			LogMsg := CONCAT('|CompId: ', WORD_TO_STRING(WsCfg.wCompId));
			LogMsg := CONCAT(LogMsg, '|WsNum: ');
			LogMsg := CONCAT(LogMsg, UINT_TO_STRING(WsCfg.iWsNum));
			LogMsg := CONCAT(LogMsg, '|Next State: ');
			LogMsg := CONCAT(LogMsg, UINT_TO_STRING(NextState));
			LogMsg := CONCAT(LogMsg,'|Cycle finished with Doc in Ws');
			Logging.Debug('FB_WsFsm.M_FinishCycle', LogMsg);	
		END_IF
	ELSIF NOT bProcessDocInWs THEN								//No document was processed before
		//switch to next state
			NextState := eWsStates.IDLE;
		IF GVL_Statemachine_ERROR_IDS.bLoggingOnOff THEN	
			LogMsg := CONCAT('|CompId: ', WORD_TO_STRING(WsCfg.wCompId));
			LogMsg := CONCAT(LogMsg, '|WsNum: ');
			LogMsg := CONCAT(LogMsg, UINT_TO_STRING(WsCfg.iWsNum));
			LogMsg := CONCAT(LogMsg, '|Next State: ');
			LogMsg := CONCAT(LogMsg, UINT_TO_STRING(NextState));
			LogMsg := CONCAT(LogMsg,'|Cycle finished without Doc in Ws');
			Logging.Debug('FB_WsFsm.M_FinishCycle', LogMsg);	
		END_IF
	ELSE														//wrong parameter Error	
		
		bMethodError := TRUE;
		
		//Throw Error		
			MethodErrorMsg.wErrorNo := GVL_Statemachine_ERROR_IDS.ERR_FSM_WRONG_INPUT_PARAMETER + GVL_Statemachine_ERROR_IDS.iErrorOffset;
			MethodErrorMsg.ErrorTyp	:= eErrorTypes._FATAL;
			M_ThrowError(	SrcState := CurrentState,
							ErrorMsg := MethodErrorMsg);	
		
		//Switch to Error state
			NextState := eWsStates.ERROR;				
	END_IF
ELSE		
		bMethodError:=TRUE;
		NextState := eWsStates.ERROR;
		
		MethodErrorMsg.wErrorNo := GVL_Statemachine_ERROR_IDS.ERR_FSM_WRONG_STATE_TO_FINISH_CYCLE + GVL_Statemachine_ERROR_IDS.iErrorOffset;
		MethodErrorMsg.ErrorTyp	:= eErrorTypes._FATAL;
		M_ThrowError(	SrcState := CurrentState,
						ErrorMsg := MethodErrorMsg);	
					
END_IF	
	
M_FinishCycle := bMethodError;
END_METHOD

METHOD PUBLIC M_ResetWs
VAR 
	LogMsg : STRING ;
END_VAR
(*
IF CurrentState <> eWsStates.IDLE THEN
	bisError := TRUE;
	bIsReset := TRUE;

END_IF
*)	
IF GVL_Statemachine_ERROR_IDS.bLoggingOnOff THEN	
	//Log data
		LogMsg := CONCAT('|CompId: ', WORD_TO_STRING(WsCfg.wCompId));
		LogMsg := CONCAT(LogMsg, '|WsNum: ');
		LogMsg := CONCAT(LogMsg, UINT_TO_STRING(WsCfg.iWsNum));
		LogMsg := CONCAT(LogMsg, '|State: ');
		LogMsg := CONCAT(LogMsg, UINT_TO_STRING(CurrentState));
		
		IF  IsValidPtr(pCurrentDoc) AND bProcessDocInWs THEN	
			LogMsg := CONCAT(LogMsg, '|DocId: ');
			LogMsg := CONCAT(LogMsg, UDINT_TO_STRING(pCurrentDoc^.ID));
		ELSE
			LogMsg := CONCAT(LogMsg, '|No doc in Ws');
		END_IF
			
		LogMsg := CONCAT(LogMsg,'|Reset was executed');
		Logging.Warn('FB_WsFsm.M_ResetWs', LogMsg);
END_IF
//Reset variables	
	CurrentState 	:= eWsStates.IDLE;
	NextState 		:= eWsStates.UNDEFINED;

	bProcessDocInWs :=FALSE; //Flag to skip cycle if there is no document in WS at machine startup. In that case the doc pointer can be invalid!
	tTimerWsProcessing(IN:=FALSE);
	pCurrentDoc := 0;
END_METHOD

METHOD PUBLIC M_ResolveErrorState : bool
VAR
	LogMsg : STRING(80);
	MethodErrorMsg : sErrorMsg;
END_VAR
MethodErrorMsg.sFunctionName := 'FB_WsFSM.M_ResolveErrorState';
MethodErrorMsg.wComponent := WsCfg.wCompId;

IF CurrentState = eWsStates.ERROR AND NextState = eWsStates.UNDEFINED THEN
	IF GVL_Statemachine_ERROR_IDS.bLoggingOnOff THEN
		//Prepare log string
			LogMsg := CONCAT('|CompId: ', WORD_TO_STRING(WsCfg.wCompId));
			LogMsg := CONCAT(LogMsg, '|WsNum: ');
			LogMsg := CONCAT(LogMsg, UINT_TO_STRING(WsCfg.iWsNum));
			LogMsg := CONCAT(LogMsg, '|Last state before error: ');		
			LogMsg := CONCAT(LogMsg, UDINT_TO_STRING(LastStateBeforeError));
			
			IF  IsValidPtr(pCurrentDoc) AND bProcessDocInWs THEN	
				LogMsg := CONCAT(LogMsg, '|DocId: ');
				LogMsg := CONCAT(LogMsg, UDINT_TO_STRING(pCurrentDoc^.ID));
			ELSE
				LogMsg := CONCAT(LogMsg, '|No doc in Ws');
			END_IF
	END_IF
	//Exclude Errors which can not be resolved
	
		CASE LastStateBeforeError OF
		
			eWsStates.IDLE :			
										IF GVL_Statemachine_ERROR_IDS.bLoggingOnOff THEN
											LogMsg := CONCAT(LogMsg,'|Error could not be resolved');
											Logging.Error('FB_WsFsm.M_ResolveErrorState', LogMsg);
										END_IF
										MethodErrorMsg.wErrorNo := GVL_Statemachine_ERROR_IDS.ERR_FSM_WORKSTATION_ERROR_CAN_NOT_BE_RESOLVED + GVL_Statemachine_ERROR_IDS.iErrorOffset;
										
										M_ThrowError(	SrcState := CurrentState,
														ErrorMsg := MethodErrorMsg);
														
			eWsStates.CYCLE_FINISHED :
										IF GVL_Statemachine_ERROR_IDS.bLoggingOnOff THEN
											LogMsg := CONCAT(LogMsg,'|Error could not be resolved');
											Logging.Error('FB_WsFsm.M_ResolveErrorState', LogMsg);
										END_IF
										MethodErrorMsg.wErrorNo := GVL_Statemachine_ERROR_IDS.ERR_FSM_WORKSTATION_ERROR_CAN_NOT_BE_RESOLVED + GVL_Statemachine_ERROR_IDS.iErrorOffset;
										
										M_ThrowError(	SrcState := CurrentState,
														ErrorMsg := MethodErrorMsg);
														
														
			ELSE //WS_PROCESSING error
				
										IF (bProcessDocInWs AND NOT IsValidPtr(pCurrentDoc)) THEN
				
											MethodErrorMsg.wErrorNo := GVL_Statemachine_ERROR_IDS.ERR_FSM_WORKSTATION_ERROR_CAN_NOT_BE_RESOLVED + GVL_Statemachine_ERROR_IDS.iErrorOffset;
																
											M_ThrowError(	SrcState := CurrentState,
															ErrorMsg := MethodErrorMsg);
															
										ELSE
											//Reset timeout timer
												tTimerWsProcessing.IN := FALSE;
												
											NextState := eWsStates.WS_PROCESSING;
											IF GVL_Statemachine_ERROR_IDS.bLoggingOnOff THEN
												LogMsg := CONCAT(LogMsg, '|Next State: ');
												LogMsg := CONCAT(LogMsg, UINT_TO_STRING(NextState));
												LogMsg := CONCAT(LogMsg,'|Error resolved successfully');
												Logging.Warn('FB_WsFsm.M_ResolveErrorState', LogMsg);
											END_IF	
										END_IF
																					
		END_CASE	
END_IF
END_METHOD

METHOD PUBLIC M_StartNewCycle : bool
VAR_INPUT
	pDocIn 			: POINTER TO sDocument;
	bProcessDoc		: BOOL;  //Flag to skip cycle if there is no document in WS at machine startup. In that case the doc pointer can be invalid!
END_VAR
VAR
	LogMsg : STRING ;
	MethodErrorMsg : sErrorMsg;
	Evt_DocIn : sDocEvent;
	bMethodError: BOOL := false;
END_VAR
MethodErrorMsg.sFunctionName := 'M_StartNewCycle';
 MethodErrorMsg.wComponent := WsCfg.wCompId;


IF CurrentState = eWsStates.IDLE  THEN
bProcessDocInWs := bProcessDoc;	

	IF  IsValidPtr(pDocIn) AND bProcessDocInWs THEN		
		
		//Set doc reference to be processed
			pCurrentDoc := pDocIn;
			
						
		//Check doc location of new doc	
		IF WsCfg.iLocation = pCurrentDoc^.Location+1 THEN				// green path - Processing of document in workstation
			//Lock document
				pCurrentDoc^.bLockedBySps := TRUE;
			
			//Set doc to not moving thus entering WS
				pCurrentDoc^.Moving := FALSE;
				
			//Set doc to WS location thus entering WS	
				pCurrentDoc^.Location := WsCfg.iLocation;
				
			//switch to next state
				NextState := eWsStates.PRE_HANDLING;
			
			//Generate OK Event
				Evt_DocIn.DocID := pCurrentDoc^.ID;
				Evt_DocIn.EventChangeFlag := switch(WsCfg.pEvt_DocIn^.EventChangeFlag);
			
			//Logging Doc Event	
				WsCfg.pEvt_DocIn^ := Evt_DocIn;
				
				IF GVL_Statemachine_ERROR_IDS.bLoggingOnOff THEN
					LogMsg := CONCAT('|CompId: ', WORD_TO_STRING(WsCfg.wCompId));
					LogMsg := CONCAT(LogMsg, '|WsNum: ');
					LogMsg := CONCAT(LogMsg, UINT_TO_STRING(WsCfg.iWsNum));
					LogMsg := CONCAT(LogMsg,'|DocIn Event written with DocId ');
					LogMsg := CONCAT(LogMsg, UDINT_TO_STRING(WsCfg.pEvt_DocIn^.DocID));
					Logging.Debug('FB_WsFsm.M_StartNewCycle', LogMsg);	
				
			
					LogMsg := CONCAT('|CompId: ', WORD_TO_STRING(WsCfg.wCompId));
					LogMsg := CONCAT(LogMsg, '|WsNum: ');
					LogMsg := CONCAT(LogMsg, UINT_TO_STRING(WsCfg.iWsNum));
					LogMsg := CONCAT(LogMsg, '|Next State: ');
					LogMsg := CONCAT(LogMsg, UINT_TO_STRING(NextState));
					LogMsg := CONCAT(LogMsg,'|Cycle started with Doc in Ws');
					Logging.Trace('FB_WsFsm.M_StartNewCycle', LogMsg);	
				END_IF
		ELSE
			
			
			MethodErrorMsg.wErrorNo := GVL_Statemachine_ERROR_IDS.ERR_FSM_WRONG_LOCATION_OF_NEW_DOC + GVL_Statemachine_ERROR_IDS.iErrorOffset;
			MethodErrorMsg.ErrorTyp	:= eErrorTypes._FATAL;			
			M_ThrowError(	SrcState := CurrentState,
							ErrorMsg := MethodErrorMsg);
										
			bMethodError:=TRUE;
			NextState := eWsStates.ERROR;
			//errorhandling wrong location of new doc!!!!
			
		END_IF
		
	ELSIF NOT bProcessDocInWs THEN	//2nd path - no document in workstation, thus skipping process
		//switch to finished state in order to skip processing
			NextState := eWsStates.CYCLE_FINISHED;
		IF GVL_Statemachine_ERROR_IDS.bLoggingOnOff THEN	
			LogMsg := CONCAT('|CompId: ', WORD_TO_STRING(WsCfg.wCompId));
			LogMsg := CONCAT(LogMsg, '|WsNum: ');
			LogMsg := CONCAT(LogMsg, UINT_TO_STRING(WsCfg.iWsNum));
			LogMsg := CONCAT(LogMsg, '|Next State: ');
			LogMsg := CONCAT(LogMsg, UINT_TO_STRING(NextState));
			LogMsg := CONCAT(LogMsg,'|Cycle started without Doc in Ws');
			Logging.Debug('FB_WsFsm.M_StartNewCycle', LogMsg);	
		END_IF
	ELSE
		//wrong parameter Error	

		
		MethodErrorMsg.wErrorNo := GVL_Statemachine_ERROR_IDS.ERR_FSM_WRONG_INPUT_PARAMETER + GVL_Statemachine_ERROR_IDS.iErrorOffset;
		MethodErrorMsg.ErrorTyp	:= eErrorTypes._FATAL;				
		M_ThrowError(	SrcState := CurrentState,
						ErrorMsg := MethodErrorMsg);

		bMethodError := TRUE;
		NextState := eWsStates.ERROR;				
	END_IF	
ELSE
	//wrong state Error
		MethodErrorMsg.wErrorNo := GVL_Statemachine_ERROR_IDS.ERR_FSM_WRONG_STATE_TO_START_NEW_CYCLE + GVL_Statemachine_ERROR_IDS.iErrorOffset;
		MethodErrorMsg.ErrorTyp	:= eErrorTypes._FATAL;			
		M_ThrowError(	SrcState := CurrentState,
						ErrorMsg := MethodErrorMsg);
		
		bMethodError := TRUE;
		NextState := eWsStates.ERROR;					
END_IF
	
	
M_StartNewCycle := bMethodError;
END_METHOD

PROPERTY PUBLIC P_bDocInWs : bool
GET
P_bDocInWs := bProcessDocInWs;
END_GET
END_PROPERTY

PROPERTY PUBLIC P_CurState : eWsStates
GET
P_CurState := CurrentState;
END_GET
END_PROPERTY

PROPERTY PUBLIC P_iDocId : udint
GET
IF IsValidPtr(pCurrentDoc) THEN
	P_iDocId := pCurrentDoc^.ID;
ELSE
	P_iDocId := 0;
END_IF
END_GET
END_PROPERTY

PROPERTY PUBLIC P_pCurDoc : Pointer to sDocument
GET
P_pCurDoc := pCurrentDoc;
END_GET
END_PROPERTY

PROPERTY PUBLIC P_tWsProcTimeout : Time
GET
P_tWsProcTimeout := WsCfg.tWsProcessingTimeout;
END_GET
SET
VAR
	LogMsg : STRING;
END_VAR
WsCfg.tWsProcessingTimeout := P_tWsProcTimeout;

//Log data
	LogMsg := CONCAT('|CompId: ', WORD_TO_STRING(WsCfg.wCompId));
	LogMsg := CONCAT(LogMsg,'|WS_PROCESSING timeout changed to: ');
	LogMsg := CONCAT(LogMsg, TIME_TO_STRING(WsCfg.tWsProcessingTimeout));
	Logging.Warn('FB_WsFsm.P_tWsProcTimeout', LogMsg);
END_SET
END_PROPERTY

METHOD PUBLIC M_CYCLE_FINISHED_DO
VAR_INPUT
END_VAR
END_METHOD

METHOD PRIVATE M_CYCLE_FINISHED_ENTRY
VAR
LogMsg : STRING;
END_VAR
//Log data
	LogMsg := CONCAT('|CompId: ', WORD_TO_STRING(WsCfg.wCompId));
	LogMsg := CONCAT(LogMsg,'|Entry of state CYCLE_FINISHED');
	Logging.Trace('FB_WsFsm.M_CYCLE_FINISHED_ENTRY', LogMsg);
END_METHOD

METHOD PRIVATE M_CYCLE_FINISHED_EXIT
VAR_INPUT
END_VAR
END_METHOD

METHOD PRIVATE M_ERROR_ENTRY
VAR
LogMsg : STRING;
END_VAR
//Log data
	LogMsg := CONCAT('|CompId: ', WORD_TO_STRING(WsCfg.wCompId));
	LogMsg := CONCAT(LogMsg,'|Entry of state ERROR');
	Logging.Trace('FB_WsFsm.M_ERROR_ENTRY', LogMsg);	
	
//bIsError := FALSE;
END_METHOD

METHOD PRIVATE M_ERROR_EXIT
END_METHOD

METHOD PRIVATE M_IDLE_DO
VAR
LogMsg : STRING;
END_VAR
END_METHOD

METHOD PRIVATE M_IDLE_ENTRY
VAR
LogMsg : STRING;
END_VAR
IF GVL_Statemachine_ERROR_IDS.bLoggingOnOff THEN
	//Log data
		LogMsg := CONCAT('|CompId: ', WORD_TO_STRING(WsCfg.wCompId));
		LogMsg := CONCAT(LogMsg,'|Entry of state IDLE');
		Logging.Trace('FB_WsFsm.M_IDLE_ENTRY', LogMsg);	
END_IF	

//bisError := FALSE;
//bIsReset := FALSE;
END_METHOD

METHOD PRIVATE M_IDLE_EXIT
VAR
LogMsg : STRING;
END_VAR
END_METHOD

METHOD PRIVATE M_INIT_WS_DO
VAR_INPUT
END_VAR
NextState := eWsStates.IDLE;
END_METHOD

METHOD PRIVATE M_INIT_WS_ENTRY
VAR_INPUT
END_VAR
END_METHOD

METHOD PRIVATE M_INIT_WS_EXIT : BOOL
VAR_INPUT
END_VAR
END_METHOD

METHOD PRIVATE M_MASTER_SYSTEM_PROCESSING_DO
VAR
	LogMsg : STRING(100);
	MethodErrorMsg : sErrorMsg;
END_VAR
//Timer will be only executed if mainfsm in running state
IF In_bPause THEN
	tTimerWsProcessing(IN := FALSE);

ELSE
	tTimerWsProcessing(IN := TRUE);
		
END_IF

//Check Relesed flag in order continue transporting
IF NOT IsValidPtr(pCurrentDoc) THEN
	MethodErrorMsg.sFunctionName := 'M_MASTER_SYSTEM_PROCESSING_DO';
	MethodErrorMsg.wComponent 	:= WsCfg.wCompId;
	MethodErrorMsg.ErrorTyp		:= eErrorTypes._FATAL;
	MethodErrorMsg.wErrorNo 	:= GVL_Statemachine_ERROR_IDS.ERR_FSM_INVALID_DOC_POINTER + GVL_Statemachine_ERROR_IDS.iErrorOffset;
	
	ErrorManagement.M_InsertNewError(MethodErrorMsg);	

	NextState := eWsStates.ERROR;			

ELSE
	IF pCurrentDoc^.Released = TRUE OR NOT pCurrentDoc^.bReleaseHandshakeActive THEN
		IF GVL_Statemachine_ERROR_IDS.bLoggingOnOff THEN
				//Logging Doc release	
					LogMsg := CONCAT('|CompId: ', WORD_TO_STRING(WsCfg.wCompId));
					LogMsg := CONCAT(LogMsg, '|WsNum: ');
					LogMsg := CONCAT(LogMsg, UINT_TO_STRING(WsCfg.iWsNum));
					LogMsg := CONCAT(LogMsg, '|DocId: ');
					LogMsg := CONCAT(LogMsg, UDINT_TO_STRING(pCurrentDoc^.ID));
					LogMsg := CONCAT(LogMsg, '|RelHndsk active: ');
					LogMsg := CONCAT(LogMsg, BOOL_TO_STRING(pCurrentDoc^.bReleaseHandshakeActive));
					
			IF pCurrentDoc^.bReleaseHandshakeActive THEN
					LogMsg := CONCAT(LogMsg,'|Release flag set to: ');
					LogMsg := CONCAT(LogMsg, BOOL_TO_STRING(pCurrentDoc^.Released));
					LogMsg := CONCAT(LogMsg,'|Proc time in ms: ');
					LogMsg := CONCAT(LogMsg, TIME_TO_STRING(tTimerWsProcessing.ET));					
			END_IF
			
			Logging.Debug('FB_WsFsm.M_MASTER_SYSTEM_PROCESSING_DO', LogMsg);
		END_IF
		NextState := eWsStates.PAST_HANDLING;
	END_IF
END_IF
END_METHOD

METHOD PRIVATE M_MASTER_SYSTEM_PROCESSING_ENTRY
VAR
	LogMsg : STRING(100);
	MethodErrorMsg : sErrorMsg;
	Evt_DocProcessStart : sDocEvent;
END_VAR

//Reset timer	
	tTimerWsProcessing(IN := FALSE, PT := WsCfg.tWsProcessingTimeout);
	
MethodErrorMsg.sFunctionName := 'M_MASTER_SYSTEM_PROCESSING_ENTRY';
MethodErrorMsg.wComponent := WsCfg.wCompId;

IF GVL_Statemachine_ERROR_IDS.bLoggingOnOff THEN
	//Log data
		LogMsg := CONCAT('|CompId: ', WORD_TO_STRING(WsCfg.wCompId));
		LogMsg := CONCAT(LogMsg,'|Entry of state MASTER_SYSTEM_PROCESSING');
		Logging.Trace('FB_WsFsm.M_MASTER_SYSTEM_PROCESSING_ENTRY', LogMsg);	
END_IF	

//Set Relesed flag in order for master system to start processing
IF NOT IsValidPtr(pCurrentDoc)  THEN
	//bIsError:=TRUE;
	MethodErrorMsg.wErrorNo := GVL_Statemachine_ERROR_IDS.ERR_FSM_INVALID_DOC_POINTER + GVL_Statemachine_ERROR_IDS.iErrorOffset;
	MethodErrorMsg.ErrorTyp	:= eErrorTypes._FATAL;				
	ErrorManagement.M_InsertNewError(MethodErrorMsg);
	NextState := eWsStates.ERROR;									

ELSIF pCurrentDoc^.bReleaseHandshakeActive THEN //sending event if flag inside ctual doc =true
	Evt_DocProcessStart.DocID := pCurrentDoc^.ID;
	Evt_DocProcessStart.EventChangeFlag := switch(WsCfg.pEvt_DocProcessStart^.EventChangeFlag);
	
	WsCfg.pEvt_DocProcessStart^ := Evt_DocProcessStart;
	
	pCurrentDoc^.Released := FALSE;
	
	IF GVL_Statemachine_ERROR_IDS.bLoggingOnOff THEN
		//Logging Doc Event	
			LogMsg := CONCAT('|CompId: ', WORD_TO_STRING(WsCfg.wCompId));
			LogMsg := CONCAT(LogMsg, '|WsNum: ');
			LogMsg := CONCAT(LogMsg, UINT_TO_STRING(WsCfg.iWsNum));
			LogMsg := CONCAT(LogMsg,'|DocProcessStart Event written with DocId ');
			LogMsg := CONCAT(LogMsg, UDINT_TO_STRING(WsCfg.pEvt_DocProcessStart^.DocID));
			LogMsg := CONCAT(LogMsg,'|Release flag set to: ');
			LogMsg := CONCAT(LogMsg, BOOL_TO_STRING(pCurrentDoc^.Released));	
			Logging.Debug('FB_WsFsm.M_MASTER_SYSTEM_PROCESSING_ENTRY', LogMsg);	
	END_IF
END_IF
END_METHOD

METHOD PRIVATE M_MASTER_SYSTEM_PROCESSING_EXIT
VAR_INPUT
END_VAR
END_METHOD

METHOD PRIVATE M_WS_PROCESSING_INTO_ERROR
VAR_INPUT
END_VAR
VAR
	LogMsg : STRING(255);
	errno : WORD;
	MethodErrorMsg : sErrorMsg;
END_VAR
MethodErrorMsg.sFunctionName := 'M_WS_PROCESSING_INTO_ERROR';
MethodErrorMsg.wComponent := WsCfg.wCompId;

IF GVL_Statemachine_ERROR_IDS.bLoggingOnOff THEN
	//----------------------------------------------------------------------------------------------------------------------------------------------------------------
	//Logging all we get	
		LogMsg := CONCAT('|CompId: ', WORD_TO_STRING(WsCfg.wCompId));
		
		LogMsg := CONCAT(LogMsg, '|WsNum: ');
		LogMsg := CONCAT(LogMsg, UINT_TO_STRING(WsCfg.iWsNum));
				
		LogMsg := CONCAT(LogMsg, '|bProcessDocInWs: ');
		LogMsg := CONCAT(LogMsg, BOOL_TO_STRING(bProcessDocInWs));
		
		LogMsg := CONCAT(LogMsg, '|Timeout: ');
		LogMsg := CONCAT(LogMsg, BOOL_TO_STRING( tTimerWsProcessing.Q AND WsCfg.tWsProcessingTimeout <> T#0S));
			
		LogMsg := CONCAT(LogMsg, '|DocId: ');
		
		IF bProcessDocInWs AND IsValidPtr(pCurrentDoc) THEN
			LogMsg := CONCAT(LogMsg, UDINT_TO_STRING(pCurrentDoc^.ID));
			
			LogMsg := CONCAT(LogMsg, '|RelHndsk active: ');
			LogMsg := CONCAT(LogMsg, BOOL_TO_STRING(pCurrentDoc^.bReleaseHandshakeActive));
			
			LogMsg := CONCAT(LogMsg, '|RelFlag: ');
			LogMsg := CONCAT(LogMsg, BOOL_TO_STRING(pCurrentDoc^.Released));
			
		ELSE
			LogMsg := CONCAT(LogMsg, 'NONE');
			
		END_IF	
	
		Logging.Debug('FB_WsFsm.M_WS_PROCESSING_INTO_ERROR', LogMsg);
END_IF	
//----------------------------------------------------------------------------------------------------------------------------------------------------------------
//Throw error

//IF NOT bIsReset THEN	//if reset => no error	
	
	IF tTimerWsProcessing.Q AND WsCfg.tWsProcessingTimeout <> T#0S THEN
		MethodErrorMsg.wErrorNo := GVL_Statemachine_ERROR_IDS.ERR_FSM_WS_PROCESSING_TIMEOUT + GVL_Statemachine_ERROR_IDS.iErrorOffset;
		
		//attach doc id to error, if one is inside ws
			IF bProcessDocInWs AND IsValidPtr(pCurrentDoc) THEN
				MethodErrorMsg.iRelatedDocId := pCurrentDoc^.ID;
				
			END_IF	

		ErrorManagement.M_InsertNewError(MethodErrorMsg);
	ELSE
		//error should be thrown already	
	
	END_IF											
//END_IF	

							
tTimerWsProcessing(IN := false);
END_METHOD

END_FUNCTION_BLOCK

// WorkstationFsm/ITF_WsFsm
INTERFACE ITF_WsFsm

METHOD PUBLIC M_ERROR_DO
END_METHOD

METHOD PUBLIC M_PAST_HANDLING_DO
VAR_OUTPUT
	bDone,
	bError : BOOL;
END_VAR
END_METHOD

METHOD PUBLIC M_PAST_HANDLING_ENTRY
END_METHOD

METHOD PUBLIC M_PAST_HANDLING_EXIT
END_METHOD

METHOD public M_PRE_HANDLING_DO
VAR_OUTPUT
	bDone,
	bError : BOOL;
END_VAR
END_METHOD

METHOD PUBLIC M_PRE_HANDLING_ENTRY
END_METHOD

METHOD PUBLIC M_PRE_HANDLING_EXIT
END_METHOD

END_INTERFACE

// WorkstationFsm/InitializeWsFsm_Base
FUNCTION InitializeWsFsm_Base : bool
VAR_INPUT
	wErrorIdOffset	: tErrorConstant;	//Offset to be added to all ErrorId´s	
	bLoggingOnOff 	: BOOL;				//TRUE => Logging activated, FALSE => Logging deactivated
END_VAR

GVL_Statemachine_ERROR_IDS.iErrorOffset 	:= wErrorIdOffset;
GVL_Statemachine_ERROR_IDS.bLoggingOnOff	:= bLoggingOnOff;

InitializeWsFsm_Base := TRUE;

END_FUNCTION
